{attribute 'qualified_only'}
{attribute 'strict'}
TYPE E_MachineMode :
(
	MODE_INITIAL := 0,
    MODE_STARTUP := 1,
    MODE_STOPPED := 2,
    MODE_RUN := 3,
    MODE_SHUTDOWN := 4,
    MODE_ESTOP := 5	
);
END_TYPE

(* stored: Version 1.1.0.1, ProductVersion 3.1.4024.16
   DUT E_MachineMode: Id {c595391c-41f4-4002-9394-719802b0de34} *)
